(* IEC 61131-3 sources: ATCMcontrol_Engineering/src/COM/softing/fc/CP/Test/Projects/WriteDialogTest, 2 files *)

(* ---- ValueTypes.ST ---- *)
(*[[
	GUID= "{D0A956E0-262A-11D2-9F4B-006008736585}"
]]*)

FUNCTION_BLOCK ValueTypes

VAR_INPUT
	varWSTRING : WSTRING;
	varTOD     : TOD;
	varDATE    : DATE;
	varDT      : DT;
	varTIME    : TIME;
	VarLREAL   : LREAL;
	varDINT    : DINT;
	varDWORD   : DWORD;
	varWORD    : WORD;
	varBYTE    : BYTE;
	varBOOL    : BOOL;
END_VAR
;
END_FUNCTION_BLOCK

(* ---- Program1.st ---- *)
(*[[
	GUID= "{D0A956BC-262A-11D2-9F4B-006008736585}"
]]*)
PROGRAM Program1

VAR
    valType : ValueTypes;
END_VAR;

END_PROGRAM
